# EPICS autosave request: alicatGasFlow/alicatGasFlow_settings.req
$(P)$(S):FLOW.HIGH
$(P)$(S):FLOW.HIHI
$(P)$(S):FLOW.LOLO
$(P)$(S):FLOW.LOW
$(P)$(S):SELECTGAS
